INTERFACE ITcoDoorCircuit

{attribute 'monitoring' := 'call'}
PROPERTY IsClosed : BOOL
GET
END_GET
END_PROPERTY

{attribute 'monitoring' := 'call'}
PROPERTY IsGlobalVoltageOk : BOOL
GET
END_GET
END_PROPERTY

{attribute 'monitoring' := 'call'}
PROPERTY IsLocalDoorsVoltageOk : BOOL
GET
END_GET
END_PROPERTY

{attribute 'monitoring' := 'call'}
PROPERTY IsLocalVoltageOk : BOOL
GET
END_GET
END_PROPERTY

{attribute 'monitoring' := 'call'}
PROPERTY IsLocked : BOOL
GET
END_GET
END_PROPERTY

{attribute 'monitoring' := 'call'}
PROPERTY IsUnLocked : BOOL
GET
END_GET
END_PROPERTY

METHOD Lock : BOOL
VAR_INPUT
END_VAR
END_METHOD

METHOD UnLock : BOOL
VAR_INPUT
END_VAR
END_METHOD

END_INTERFACE

(* stored: Version 1.1.0.1
   Itf ITcoDoorCircuit: Id {5c977ebf-d143-4a1d-af86-7e0c865d113b}
   Property IsClosed: Id {d88ee396-761e-4092-ba7a-fed7e19f766d}
   Get Get: Id {03410a06-1561-4c41-be76-b5d9d0cb1905}
   Property IsGlobalVoltageOk: Id {128a1fcf-069f-4dec-872c-34d8079803e8}
   Get Get: Id {7de0b1e8-0f12-46b6-9fdf-1a33d0365744}
   Property IsLocalDoorsVoltageOk: Id {806b6911-d960-4ee7-a26b-d21d53ef3bcb}
   Get Get: Id {dbd706b2-1e39-4236-a088-ce62ca38840f}
   Property IsLocalVoltageOk: Id {26e9c345-b9ea-4e2a-948b-2cc709e498a8}
   Get Get: Id {9f033ff7-9ef1-4364-8b1f-1479ed367351}
   Property IsLocked: Id {38c4456d-9c42-4303-9e74-71242df9ef2a}
   Get Get: Id {d037bb63-5b4e-44a7-b334-f58ab6995686}
   Property IsUnLocked: Id {5cffd108-0736-459c-9646-721a79d55fbb}
   Get Get: Id {ef4ffdc0-cdc8-43a7-84ff-5d86ac874173}
   Method Lock: Id {80d281cb-ac8f-4233-8ff4-b9be85944670}
   Method UnLock: Id {b0c2b8c9-b76e-4208-ace2-1e2fb1791f22} *)
